// SIMATIC S7-200 SMART project (STEP 7-Micro/WIN SMART), CPU ST60

SYMBOL_TABLE Table 1
FOR_PULSE        M20.0
GLASS_SUCK       M10.1
AUTO_COIL        M10.0
CYL_DN_MEM_BITS  M0.7
READY_COIL       M0.6
REV_COIL         M0.5
FAWARD_COIL      M0.4
SUCK_COIL        M0.3
AUTO_SEL         M0.1
MAN_SEL          M0.0
END_SYMBOL_TABLE

SYMBOL_TABLE System Symbols
Always_On        SM0.0    // Always ON
END_SYMBOL_TABLE

ORGANIZATION_BLOCK MAIN:OB1
TITLE=MHSF 
BEGIN
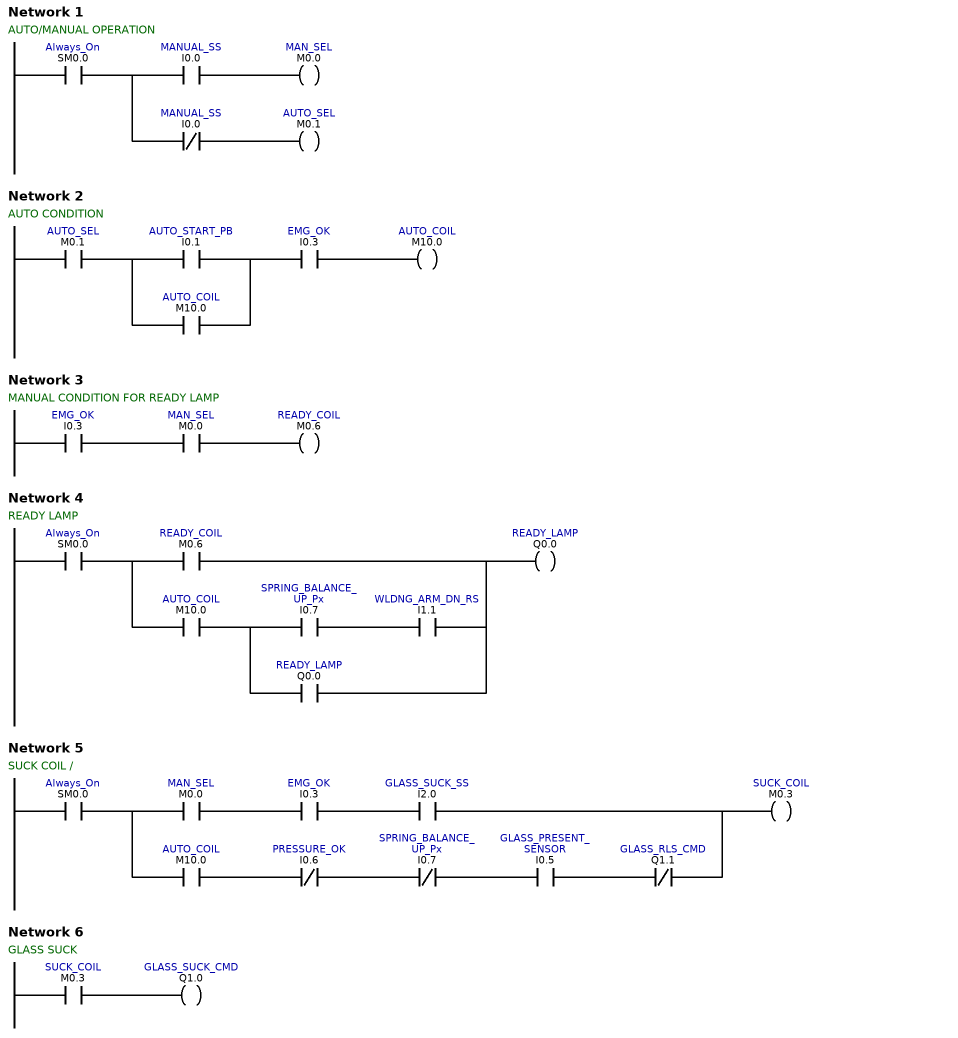
Network 1
// AUTO/MANUAL OPERATION 
LD     Always_On:SM0.0
LPS
A      MANUAL_SS:I0.0
=      MAN_SEL:M0.0
LPP
AN     MANUAL_SS:I0.0
=      AUTO_SEL:M0.1
Network 2
// AUTO CONDITION 
LD     AUTO_SEL:M0.1
LD     AUTO_START_PB:I0.1
O      AUTO_COIL:M10.0
ALD
A      EMG_OK:I0.3
=      AUTO_COIL:M10.0
Network 3
// MANUAL CONDITION FOR READY LAMP
LD     EMG_OK:I0.3
A      MAN_SEL:M0.0
=      READY_COIL:M0.6
Network 4
// READY LAMP 
LD     Always_On:SM0.0
LD     READY_COIL:M0.6
LD     AUTO_COIL:M10.0
LD     SPRING_BALANCE_UP_Px:I0.7
A      WLDNG_ARM_DN_RS:I1.1
O      READY_LAMP:Q0.0
ALD
OLD
ALD
=      READY_LAMP:Q0.0
Network 5
// SUCK COIL
// 
LD     Always_On:SM0.0
LD     MAN_SEL:M0.0
A      EMG_OK:I0.3
A      GLASS_SUCK_SS:I2.0
LD     AUTO_COIL:M10.0
AN     PRESSURE_OK:I0.6
AN     SPRING_BALANCE_UP_Px:I0.7
A      GLASS_PRESENT_SENSOR:I0.5
AN     GLASS_RLS_CMD:Q1.1
OLD
ALD
=      SUCK_COIL:M0.3
Network 6
// GLASS SUCK
LD     SUCK_COIL:M0.3
=      GLASS_SUCK_CMD:Q1.0
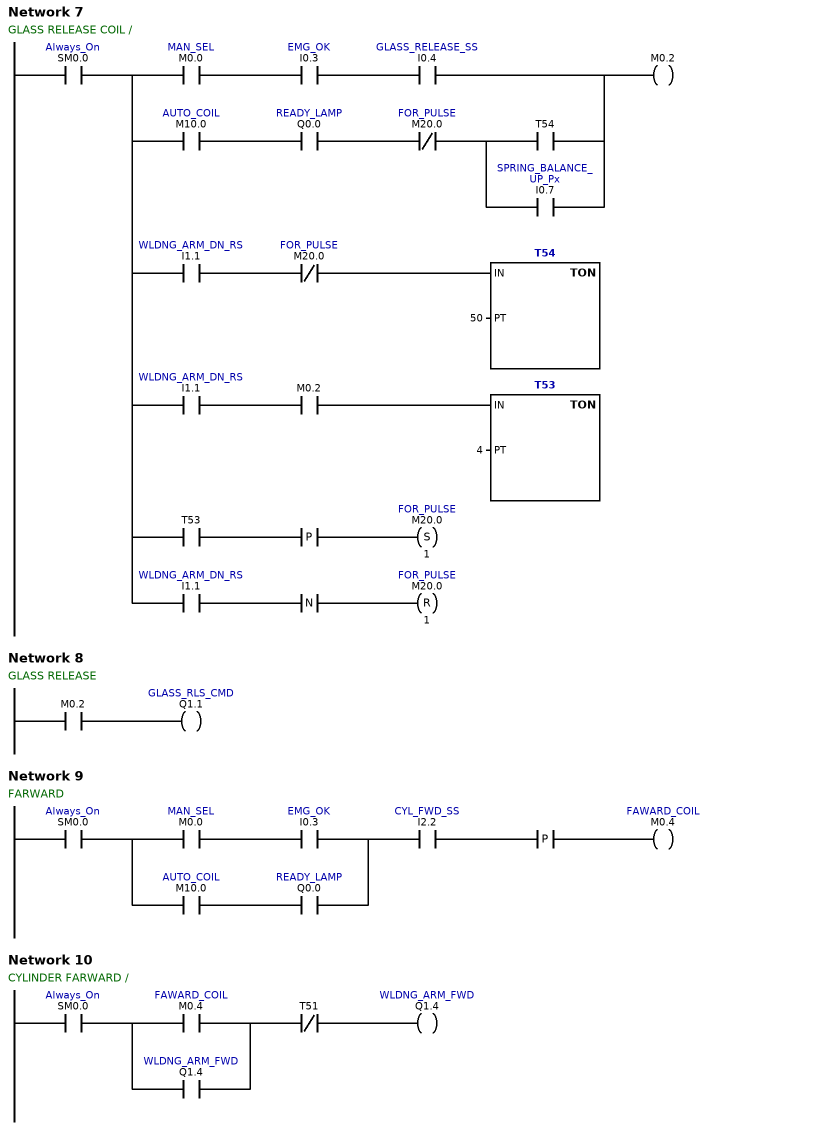
Network 7
// GLASS RELEASE COIL
// 
LD     Always_On:SM0.0
LPS
LD     MAN_SEL:M0.0
A      EMG_OK:I0.3
A      GLASS_RELEASE_SS:I0.4
LD     AUTO_COIL:M10.0
A      READY_LAMP:Q0.0
AN     FOR_PULSE:M20.0
LD     T54
O      SPRING_BALANCE_UP_Px:I0.7
ALD
OLD
ALD
=      M0.2
LPP
LPS
A      WLDNG_ARM_DN_RS:I1.1
AN     FOR_PULSE:M20.0
TON    T54, 50
LRD
A      WLDNG_ARM_DN_RS:I1.1
A      M0.2
TON    T53, 4
LRD
A      T53
EU
S      FOR_PULSE:M20.0, 1
LPP
A      WLDNG_ARM_DN_RS:I1.1
ED
R      FOR_PULSE:M20.0, 1
Network 8
// GLASS RELEASE
LD     M0.2
=      GLASS_RLS_CMD:Q1.1
Network 9
// FARWARD
LD     Always_On:SM0.0
LD     MAN_SEL:M0.0
A      EMG_OK:I0.3
LD     AUTO_COIL:M10.0
A      READY_LAMP:Q0.0
OLD
ALD
A      CYL_FWD_SS:I2.2
EU
=      FAWARD_COIL:M0.4
Network 10
// CYLINDER FARWARD
// 
LD     Always_On:SM0.0
LD     FAWARD_COIL:M0.4
O      WLDNG_ARM_FWD:Q1.4
ALD
AN     T51
=      WLDNG_ARM_FWD:Q1.4
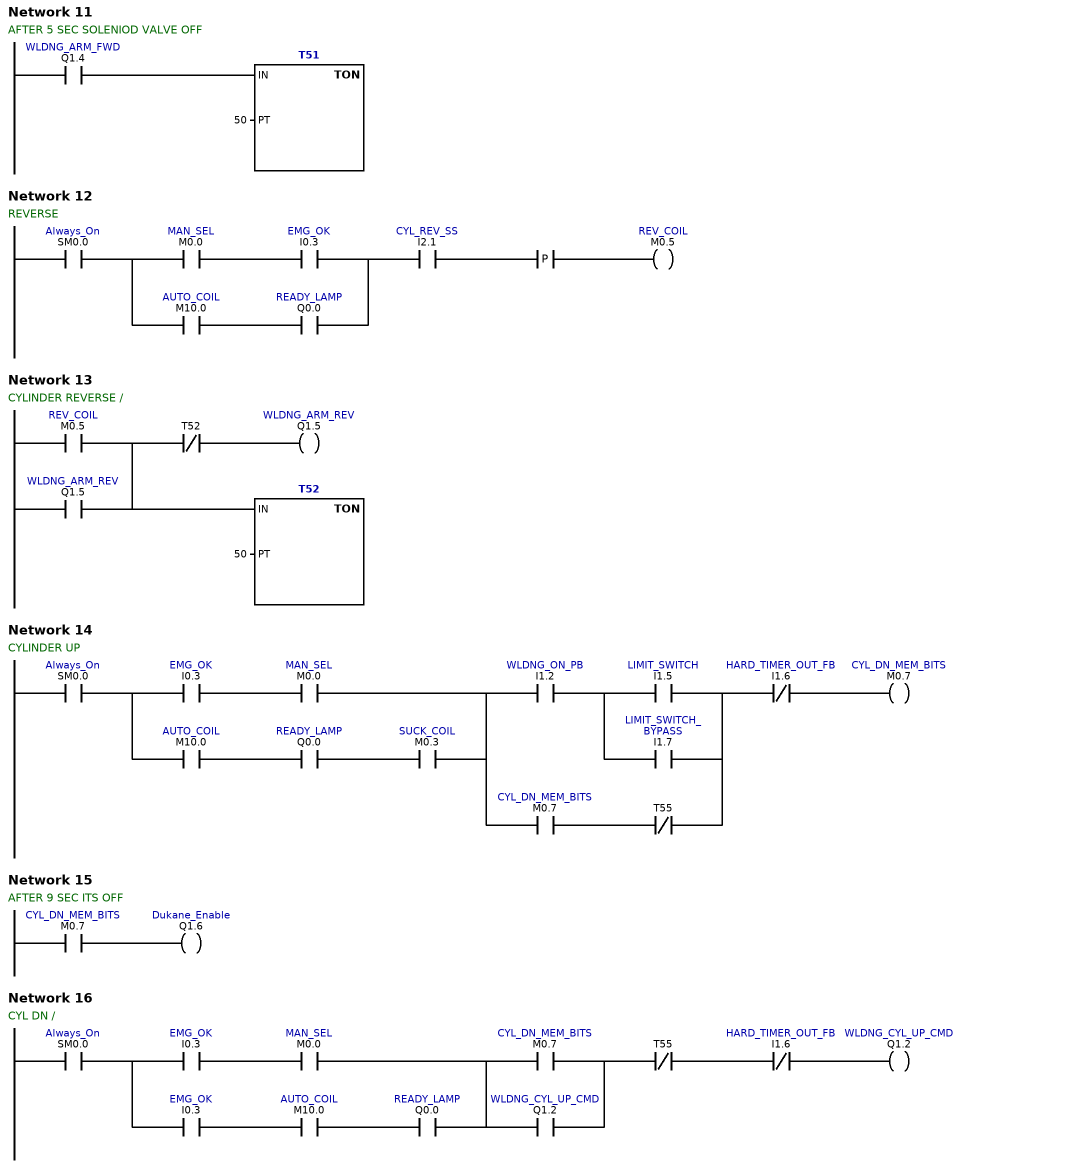
Network 11
// AFTER 5 SEC SOLENIOD VALVE OFF
LD     WLDNG_ARM_FWD:Q1.4
TON    T51, 50
Network 12
// REVERSE
LD     Always_On:SM0.0
LD     MAN_SEL:M0.0
A      EMG_OK:I0.3
LD     AUTO_COIL:M10.0
A      READY_LAMP:Q0.0
OLD
ALD
A      CYL_REV_SS:I2.1
EU
=      REV_COIL:M0.5
Network 13
// CYLINDER REVERSE
// 
LD     REV_COIL:M0.5
O      WLDNG_ARM_REV:Q1.5
LPS
AN     T52
=      WLDNG_ARM_REV:Q1.5
LPP
TON    T52, 50
Network 14
// CYLINDER UP
LD     Always_On:SM0.0
LD     EMG_OK:I0.3
A      MAN_SEL:M0.0
LD     AUTO_COIL:M10.0
A      READY_LAMP:Q0.0
A      SUCK_COIL:M0.3
OLD
ALD
LD     WLDNG_ON_PB:I1.2
LD     LIMIT_SWITCH:I1.5
O      LIMIT_SWITCH_BYPASS:I1.7
ALD
LD     CYL_DN_MEM_BITS:M0.7
AN     T55
OLD
ALD
AN     HARD_TIMER_OUT_FB:I1.6
=      CYL_DN_MEM_BITS:M0.7
Network 15
// AFTER 9 SEC ITS OFF
LD     CYL_DN_MEM_BITS:M0.7
=      Dukane_Enable:Q1.6
Network 16
// CYL DN
// 
LD     Always_On:SM0.0
LD     EMG_OK:I0.3
A      MAN_SEL:M0.0
LD     EMG_OK:I0.3
A      AUTO_COIL:M10.0
A      READY_LAMP:Q0.0
OLD
ALD
LD     CYL_DN_MEM_BITS:M0.7
O      WLDNG_CYL_UP_CMD:Q1.2
ALD
AN     T55
AN     HARD_TIMER_OUT_FB:I1.6
=      WLDNG_CYL_UP_CMD:Q1.2
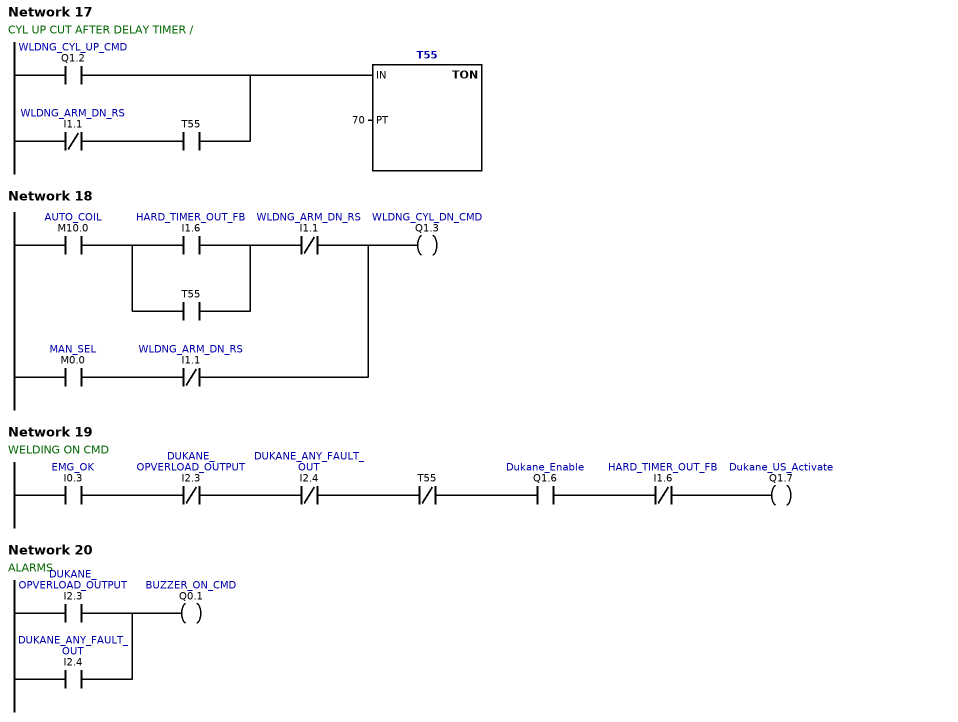
Network 17
// CYL UP CUT AFTER DELAY TIMER
// 
LD     WLDNG_CYL_UP_CMD:Q1.2
LDN    WLDNG_ARM_DN_RS:I1.1
A      T55
OLD
TON    T55, 70
Network 18
LD     AUTO_COIL:M10.0
LD     HARD_TIMER_OUT_FB:I1.6
O      T55
ALD
AN     WLDNG_ARM_DN_RS:I1.1
LD     MAN_SEL:M0.0
AN     WLDNG_ARM_DN_RS:I1.1
OLD
=      WLDNG_CYL_DN_CMD:Q1.3
Network 19
// WELDING ON CMD
LD     EMG_OK:I0.3
AN     DUKANE_OPVERLOAD_OUTPUT:I2.3
AN     DUKANE_ANY_FAULT_OUT:I2.4
AN     T55
A      Dukane_Enable:Q1.6
AN     HARD_TIMER_OUT_FB:I1.6
=      Dukane_US_Activate:Q1.7
Network 20
// ALARMS
LD     DUKANE_OPVERLOAD_OUTPUT:I2.3
O      DUKANE_ANY_FAULT_OUT:I2.4
=      BUZZER_ON_CMD:Q0.1
END_ORGANIZATION_BLOCK
